{attribute addProperty BoxType "EL3681-0000-0020"}
{attribute addProperty Id "SAI_InputsAT %I*SAI_Inputs_166EE3574860SAI_RangeAT %I*SAI_Range_DF9848341620SAI_Range_1AT %Q*SAI_Range_80D0ED7D1620WcStateAT %I*WcState_98A4DF7520.250InfoDataAT %I*InfoData_BC63D37F80100"}
{attribute addProperty CRC "2173550029"}
{attribute addProperty SizeInBites "162"}
{attribute addProperty SizeInBytes "20.25"}
TYPE EL3681_C596F5D1 :
STRUCT
	{attribute addProperty Name "SAI_Inputs"}
	SAI_Inputs : SAI_Inputs_166EE357;
	{attribute addProperty Name "SAI_Range"}
	SAI_Range : SAI_Range_DF984834;
	{attribute addProperty Name "SAI_Range_1"}
	SAI_Range_1 : SAI_Range_80D0ED7D;
	{attribute addProperty Name "WcState"}
	WcState : WcState_98A4DF75;
	{attribute addProperty Name "InfoData"}
	InfoData : InfoData_BC63D37F;
END_STRUCT
END_TYPE

(* stored: Version 1.2.0.0, ProductVersion 3.1.4024.9
   DUT EL3681_C596F5D1: Id {27ba6d90-598e-4f5f-9f8a-326c894f4c3a} *)
